{attribute 'linkalways'} 
{attribute 'no_explicit_call' := 'This FB is a CLASS and must be accessed using methods or properties'}
{attribute 'enable_dynamic_creation'}
FUNCTION_BLOCK FINAL EQ_SINT EXTENDS Node
VAR
	in1 : _SINT(0);
	in2 : _SINT(0);
	out : _BOOL(FALSE);
END_VAR

METHOD PUBLIC Clone : I_Node
VAR
	pNode : POINTER TO EQ_SINT;
END_VAR
pNode := __NEW(EQ_SINT);
Clone := pNode^;
END_METHOD

METHOD FB_init : BOOL
VAR_INPUT
	bInitRetains : BOOL; // if TRUE, the retain variables are initialized (warm start / cold start)
	bInCopyCode : BOOL;  // if TRUE, the instance afterwards gets moved into the copy code (online change)
END_VAR
AddInput('in1',THIS^.in1);
AddInput('in2',THIS^.in2);
AddOutput('out', THIS^.out);
END_METHOD

METHOD PROTECTED OnExecute
VAR
END_VAR
out.Value := in1.Value = in2.Value;
END_METHOD

END_FUNCTION_BLOCK

(* stored: Version 1.1.0.1, ProductVersion 3.1.4024.15
   POU EQ_SINT: Id {7d931abc-cb39-4e45-a56d-1ac48f46a1c9}, SpecialFunc None
   Folder Constructor: Id {443513e4-4659-4e50-b6b2-a88bd0654b82}
   Method Clone: Id {84cee125-0fd8-4220-b3c1-d41c6c8a722d}
   Method FB_init: Id {6797a4b9-c097-40b7-8232-0de6707b6453}
   Method OnExecute: Id {d3dbb164-fde0-490d-bbcc-e5aaceef55d1} *)
